(* IEC 61131-3 sources: generating_plc_code_with_llms/Code#1/Bard/third run, 21 files *)

(* ---- 14.st ---- *)
// 9.13s
// 2
FUNCTION FC1001(current_value: REAL, switching_value: REAL, hysteresis_percent: REAL): BOOL;
VAR
  previous_value: REAL;
  hysteresis_value: REAL;
  output_state: BOOL;

BEGIN

  // Initialize variables on first call
  IF NOT FC1001_initialized THEN
    previous_value := current_value;
    FC1001_initialized := TRUE;
  END_IF;

  // Calculate hysteresis value
  hysteresis_value := switching_value * hysteresis_percent / 100.0;

  // Determine output state based on current value and hysteresis
  IF current_value > switching_value + hysteresis_value THEN
    output_state := TRUE;
  ELSIF current_value < switching_value - hysteresis_value THEN
    output_state := FALSE;
  ELSE
    output_state := previous_value; // Maintain previous state to prevent fluttering
  END_IF;

  // Update previous value for next call
  previous_value := current_value;

  FC1001 := output_state;
END_FUNCTION

(* ---- 15.st ---- *)
// 12.79s
// 2
FUNCTION FC1002(E_A: BOOL, ultrasonic_presence: BOOL, P_HU: BOOL, P_AL: BOOL, P1: BOOL):
VAR
  monitoring_active: BOOL;
  presence_detected: BOOL;
  presence_timer: TIME;

BEGIN

  // Determine monitoring activation based on switch E_A
  monitoring_active := E_A;

  // Update presence_detected based on ultrasonic_presence and monitoring_active
  IF monitoring_active THEN
    IF ultrasonic_presence THEN
      presence_detected := TRUE;
    ELSIF NOT presence_detected THEN
      TOF(IN := TRUE, PT := #3000ms, Q := presence_timer);
    ELSE
      IF presence_timer.ET THEN
        presence_detected := FALSE;
      END_IF;
    END_IF;
  ELSE
    presence_detected := FALSE;
  END_IF;

  // Set output signals based on presence_detected and monitoring_active
  P_HU := monitoring_active AND presence_detected;
  P_AL := monitoring_active AND presence_detected AND presence_timer.ET;
  P1 := monitoring_active;

  FC1002 := (monitoring_active, presence_detected);
END_FUNCTION

(* ---- 18.st ---- *)
// 6.4s
// 2
FUNCTION FC1003(IN: REAL; IN_MIN: REAL; IN_MAX: REAL; OUT_MIN: REAL; OUT_MAX: REAL): REAL;

VAR
  range_factor: REAL;
  scaled_value: REAL;

BEGIN

  // Calculate range factor
  range_factor := (OUT_MAX - OUT_MIN) / (IN_MAX - IN_MIN);

  // Scale input value
  scaled_value := IN - IN_MIN;

  // Convert scaled value to output range
  FC1003 := scaled_value * range_factor + OUT_MIN;

  RETURN FC1003;
END_FUNCTION

(* ---- 19.st ---- *)
// 8.77s
// 2
FUNCTION_BLOCK FB1005

VAR
  START: BOOL;
  THICKNESS: BYTE;
  V_MAX: REAL;
  V_MIN: REAL;
  D_MAX: BYTE;
  D_MIN: BYTE;

  M_MAX: REAL;
  M_MIN: REAL;
  reject: BOOL;

BEGIN

  // Initialize variables
  M_MAX := 0.0;
  M_MIN := 0.0;
  reject := FALSE;

  // Read start signal
  START := SensorS1;

  // Read thickness
  THICKNESS := MD_1;

  // Check for new measurement
  IF START AND NOT reject THEN
    // Reset reject flag and minimum and maximum thickness values
    reject := FALSE;
    M_MAX := 0.0;
    M_MIN := 0.0;

    // Calculate thickness from laser measurements
    M_MAX := laser_measurement1 - laser_measurement2;

    // Check if thickness is outside tolerance
    IF M_MAX > V_MAX OR M_MAX < V_MIN THEN
      reject := TRUE;
      P1 := TRUE;
    END_IF;

    // Update minimum thickness value
    IF M_MIN = 0.0 OR M_MIN > M_MAX THEN
      M_MIN := M_MAX;
    END_IF;
  END_IF;

  // Write maximum thickness value to output
  D_MAX := INT(M_MAX);

  // Write minimum thickness value to output
  D_MIN := INT(M_MIN);

END_FUNCTION_BLOCK

(* ---- 21.st ---- *)
// 13.61s
// 2
FUNCTION_BLOCK BURNER

VAR
IN: BOOL;             // Start signal
OVER_TEMP: BOOL;      // Boiler thermostat protection
OIL_TEMP: BOOL;       // Oil temperature signal
STAGE2: BOOL;        // Second stage activation
RST: BOOL;            // Reset signal
STATUS: INT;       // Status output (110-Standby, 111-Startup, 112-Stage 1, 113-Stage 2)
ERROR: INT;         // Error output (0-No error, 1-Oil warming timeout, 2-Flame during pre-heat, ...)

internal_state: INT; // Internal state machine variable
timer_preheat: TIME;  // Timer for pre-heating
timer_prevent: TIME;  // Timer for pre-ventilation
timer_safety: TIME;   // Timer for flame safety
timer_post_ignit: TIME; // Timer for post-ignition delay
timer_stage2: TIME;   // Timer for stage 2 delay
timer_lockout: TIME;  // Timer for lockout

BEGIN

// Initialize variables
internal_state := 110; // Standby
timer_preheat := 0s;
timer_prevent := 0s;
timer_safety := 0s;
timer_post_ignit := 0s;
timer_stage2 := 0s;
timer_lockout := 0s;
STATUS := 110;
ERROR := 0;

// Main loop
WHILE TRUE DO

// Check for reset
IF RST THEN
  IF timer_lockout.ET THEN
    internal_state := 110;
    STATUS := 110;
    ERROR := 0;
  END_IF;
ELSE

  // Check overall conditions
  IF OVER_TEMP THEN
    internal_state := 110;
    STATUS := 110;
    ERROR := 9;
  ELSIF internal_state = 110 AND IN THEN
    internal_state := 111;
    STATUS := 111;
  END_IF;

  // State machine
  CASE internal_state OF
    111: // Startup sequence
      TOF(IN := TRUE, PT := #PRE_HEAT_TIME, Q := timer_preheat);
      IF OIL_TEMP AND timer_preheat.ET THEN
        internal_state := 112;
        STATUS := 112;
        timer_prevent := 0s;
      ELSIF timer_preheat.ET THEN
        internal_state := 110;
        STATUS := 110;
        ERROR := 1;
      END_IF;
    112: // Stage 1 operation
      TOF(IN := TRUE, PT := #PRE_VENTILATION_TIME, Q := timer_prevent);
      IF timer_prevent.ET THEN
        TOF(IN := TRUE, PT := #PRE_IGNITE_TIME, Q := timer_post_ignit);
        TOF(IN := TRUE, PT := #SAFETY_TIME, Q := timer_safety);
        IF (TIMER_IGNITION_ACTIVE) THEN
          ERROR := 2;
        ELSIF NOT TIMER_FLAME_DETECTED THEN
          ERROR := 4;
        ELSIF timer_safety.ET THEN
          internal_state := 112; // Restart ignition
          timer_post_ignit := 0s;
        ELSE
          TOF(IN := TRUE, PT := #POST_IGNITE_TIME, Q := timer_post_ignit);
          IF timer_post_ignit.ET AND NOT TIMER_FLAME_DETECTED THEN
            ERROR := 5;
          ELSE
            timer_stage2 := #STAGE2_DELAY;
          END_IF;
        END_IF;
      END_IF;
    113: // Stage 2 operation
      TOF(IN := TRUE, PT := timer_stage2, Q := timer_stage2);
      IF STAGE2 AND timer_stage2.ET THEN
        internal_state := 113; // Continue in stage 2
        timer_stage2 := 0s;
      ELSEIF NOT TIMER_FLAME_DETECTED OR MULTIPLE_IGNITION THEN
        internal_state := 112; // Restart ignition
// 23.8s
      ELSEIF NOT TIMER_FLAME_DETECTED OR MULTIPLE_IGNITION THEN
        internal_state := 112; // Restart ignition
        timer_post_ignit := 0s;
      END_IF;
    END_CASE;

    // Lockout timer
  TOF(IN := TRUE, PT := #LOCKOUT_TIME, Q := timer_lockout);

END_IF;

END_WHILE;

END_FUNCTION_BLOCK

(* ---- 1.st ---- *)
//5.95s
//3
PROGRAM MyProgram

VAR
  xAlarm1: BOOL;
  xAlarm2: BOOL;
  xAllOn: BOOL;
  xAllOff: BOOL;

BEGIN

  IF xAllOn THEN
    xAlarm1 := TRUE;
    xAlarm2 := TRUE;
  ELSIF xAllOff THEN
    xAlarm1 := FALSE;
    xAlarm2 := FALSE;
  ELSE
    // Process alarm conditions
  END_IF;

END_PROGRAM

(* ---- 10.st ---- *)
//7.98s
// 2
PROGRAM SigmoidFunction

VAR
  x: REAL;
  y: REAL;

FUNCTION Sigmoid(x: REAL): REAL;
  BEGIN
    y := 1.0 / (1.0 + Exp(-x));
    Sigmoid := y;
  END_FUNCTION;

BEGIN
  x := 1.0;
  y := Sigmoid(x);
END_PROGRAM

(* ---- 11.st ---- *)
//6.85s
// 2
PROGRAM SignFunction

VAR
  x: REAL;
  y: REAL;

FUNCTION Sign(x: REAL): REAL;
  BEGIN
    IF x > 0 THEN
      y := 1.0;
    ELSIF x < 0 THEN
      y := -1.0;
    ELSE
      y := 0.0;
    END_IF;
    Sign := y;
  END_FUNCTION;

BEGIN
  x := 1.0;
  y := Sign(x);
END_PROGRAM

(* ---- 12.st ---- *)
//8.86s
// 2
PROGRAM HyperbolicSine

VAR
x: REAL;
y: REAL;

FUNCTION Sinh(x: REAL): REAL;
BEGIN
y := (Exp(x) - Exp(-x)) / 2.0;
Sinh := y;
END_FUNCTION;

BEGIN
x := 1.0;
y := Sinh(x);
END_PROGRAM;

(* ---- 13.st ---- *)
//12.15s
// 2
PROGRAM NumberSearch

VAR
  numbers: ARRAY[0..99] OF INT;
  targetNumber: INT := 10;
  found: BOOL := FALSE;
  index: INT;

BEGIN

  // Initialize the list with random numbers
  FOR index := 0 TO 99 DO
    numbers[index] := RANDOM(1, 100);
  END_FOR;

  index := 0;

  REPEAT
    IF numbers[index] = targetNumber THEN
      found := TRUE;
      EXIT;
    END_IF;

    index := index + 1;
  UNTIL index = 100;

  // Handle the result
  IF found THEN
    WRITE_STRING('The number ' + STRING(targetNumber) + ' was found at index ' + STRING(index));
  ELSE
    WRITE_STRING('The number ' + STRING(targetNumber) + ' was not found in the list');
  END_IF;

END_PROGRAM

(* ---- 16.st ---- *)
//13.09s
// 2
PROGRAM TrafficLight

VAR
  North_green: BOOL;
  North_yellow: BOOL;
  North_red: BOOL;
  East_green: BOOL;
  East_yellow: BOOL;
  East_red: BOOL;
  timer: TIME;

BEGIN

  // Initialize all lights to red
  North_green := FALSE;
  North_yellow := FALSE;
  North_red := TRUE;
  East_green := FALSE;
  East_yellow := FALSE;
  East_red := TRUE;

  // Start the timer
  TON(IN := TRUE, PT := #10000ms, Q := timer);

  WHILE TRUE DO
    // Check the timer value and set the light signals accordingly
    IF timer.ET THEN
      // North light green
      North_green := TRUE;
      North_yellow := FALSE;
      North_red := FALSE;
      East_green := FALSE;
      East_yellow := FALSE;
      East_red := TRUE;

      // Wait for 5000ms
      DELAY(5000);

      // North light yellow
      North_green := FALSE;
      North_yellow := TRUE;
      North_red := FALSE;
      East_green := FALSE;
      East_yellow := FALSE;
      East_red := TRUE;

      // Wait for 500ms
      DELAY(500);

      // North light red, East light green
      North_green := FALSE;
      North_yellow := FALSE;
      North_red := TRUE;
      East_green := TRUE;
      East_yellow := FALSE;
      East_red := FALSE;

      // Wait for 4000ms
      DELAY(4000);

      // East light yellow
      North_green := FALSE;
      North_yellow := FALSE;
      North_red := TRUE;
      East_green := FALSE;
      East_yellow := TRUE;
      East_red := FALSE;

      // Wait for 500ms
      DELAY(500);

      // Reset the timer
      TOF(IN := timer.Q, PT := #10000ms, Q := timer);
    END_IF;
  END_WHILE;

END_PROGRAM

(* ---- 17.st ---- *)
//11.4s
// 2
PROGRAM WeatherStation

VAR
  temperatureAnalogValue: INT; // Temperature analog input value
  temperaturePercent: REAL; // Temperature converted to percent
  humidity: INT; // Humidity analog input value
  humidityPercent: REAL; // Humidity converted to percent
  temperatureText: STRING(10); // Text representation of temperature
  overallText: STRING(10); // Overall assessment of temperature and humidity

BEGIN

  // Read temperature analog value
  temperatureAnalogValue := ReadAnalogInput(TemperatureAnalogInputChannel);

  // Convert temperature analog value to percent
  temperaturePercent := REAL(temperatureAnalogValue) / 32767.0 * 100.0;

  // Evaluate temperature and set temperature text
  IF temperaturePercent < 18.0 THEN
    temperatureText := 'Cold';
  ELSIF temperaturePercent <= 25.0 THEN
    temperatureText := 'Opt';
  ELSE
    temperatureText := 'Hot';
  END_IF;

  // Read humidity analog value
  humidity := ReadAnalogInput(HumidityAnalogInputChannel);

  // Convert humidity analog value to percent
  humidityPercent := REAL(humidity) / 32767.0 * 100.0;

  // Evaluate humidity and temperature
  IF 40.0 <= humidityPercent <= 75.0 AND 18.0 <= temperaturePercent <= 25.0 THEN
    overallText := 'Opt';
  ELSE
    overallText := 'Temp. OK';
  END_IF;

  // Display temperature and humidity
  WRITE_STRING('Temperature: ' + STRING(temperaturePercent) + '% - ' + temperatureText);
  WRITE_STRING('Humidity: ' + STRING(humidityPercent) + '% - ' + overallText);

END_PROGRAM

(* ---- 2.st ---- *)
//4.63s
//2
PROGRAM BinomialCoefficient

VAR
  n: INT;
  k: INT;
  result: INT;

BEGIN

  IF k > n OR k < 0 THEN
    result := 0;
  ELSIF k = 0 OR k = n THEN
    result := 1;
  ELSE
    result := BinomialCoefficient(n - 1, k - 1) + BinomialCoefficient(n - 1, k);
  END_IF;
END_PROGRAM

(* ---- 20.st ---- *)
// 8.08s
// 2
PROGRAM Interlock

VAR
  I1: BOOL;
  I2: BOOL;
  Q1: BOOL;
  Q2: BOOL;
  Q1Timer: TIME;
  Q2Timer: TIME;

BEGIN

  // Initialize timers
  Q1Timer := 0.0s;
  Q2Timer := 0.0s;

  WHILE TRUE DO
    // Check input I1
    IF I1 THEN
      // Enable timer for Q1
      TOF(IN := TRUE, PT := #TL, Q := Q1Timer);

      // Set output Q1
      Q1 := TRUE;

      // Reset output Q2
      Q2 := FALSE;

      // Clear Q2 timer
      Q2Timer := 0.0s;
    END_IF;

    // Check input I2
    IF I2 THEN
      // Enable timer for Q2
      TOF(IN := TRUE, PT := #TL, Q := Q2Timer);

      // Set output Q2
      Q2 := TRUE;

      // Reset output Q1
      Q1 := FALSE;

      // Clear Q1 timer
      Q1Timer := 0.0s;
    END_IF;

    // Check if Q2 can be enabled
    IF Q2Timer > TL AND NOT Q2 THEN
      // Enable Q2
      Q2Timer := 0.0s;

      Q2 := TRUE;
    END_IF;

    // Check if Q1 can be enabled
    IF Q1Timer > TL AND NOT Q1 THEN
      // Enable Q1
      Q1Timer := 0.0s;

      Q1 := TRUE;
    END_IF;
  END_WHILE;

END_PROGRAM

(* ---- 3.st ---- *)
//10.15s
// 2
PROGRAM Fibonacci

VAR
  n: INT;
  result: INT;

FUNCTION Fibonacci(n: INT): INT;
VAR
  a: INT;
  b: INT;
  i: INT;

BEGIN
  a := 0;
  b := 1;

  FOR i := 1 TO n DO
    result := a + b;
    a := b;
    b := result;
  END_FOR;

  Fibonacci := result;
END_FUNCTION;

BEGIN
  n := 10;
  result := Fibonacci(n);
END_PROGRAM

(* ---- 4.st ---- *)
//7.39s
// 2
PROGRAM FillLevelCheck

VAR
  fillLevelAnalogValue: INT;
  fillLevelPercent: REAL;
  lowLevelOutput: BOOL;
  okLevelOutput: BOOL;
  highLevelOutput: BOOL;
  warningHornOutput: BOOL;

BEGIN

  // Read the fill level analog value
  fillLevelAnalogValue := ReadAnalogInput(AnalogInputChannel);

  // Convert the analog value to a percentage
  fillLevelPercent := REAL(fillLevelAnalogValue) / 32767.0 * 100.0;

  // Check the fill level and set the output variables accordingly
  CASE fillLevelPercent OF
    0.0 TO 1.0:
      lowLevelOutput := TRUE;
      okLevelOutput := FALSE;
      highLevelOutput := FALSE;
      warningHornOutput := TRUE;
    1.0 TO 90.0:
      lowLevelOutput := FALSE;
      okLevelOutput := TRUE;
      highLevelOutput := FALSE;
      warningHornOutput := FALSE;
    90.0 TO 100.0:
      lowLevelOutput := FALSE;
      okLevelOutput := FALSE;
      highLevelOutput := TRUE;
      warningHornOutput := FALSE;
    ELSE:
      // Invalid fill level
  END_CASE;

  // Write the output variables to the outputs
  WriteDigitalOutput(LowLevelOutputChannel, lowLevelOutput);
  WriteDigitalOutput(OkLevelOutputChannel, okLevelOutput);
  WriteDigitalOutput(HighLevelOutputChannel, highLevelOutput);
  WriteDigitalOutput(WarningHornOutputChannel, warningHornOutput);

END_PROGRAM

(* ---- 5.st ---- *)
//10.45s
// 2
PROGRAM GateController

VAR
  Start_Loop: BOOL;
  Gate_Open: BOOL;
  App_Or_Car_Sensed: BOOL;
  Auth_String: STRING(10);
  One_Hour_Timer: TIME;

BEGIN

  // Check if the start loop signal is active
  IF Start_Loop THEN
    // Start the one-hour timer
    TON(IN := TRUE, PT := #1H, Q := One_Hour_Timer);

    // Check if the gate is open and the timer has timed out
    IF Gate_Open AND One_Hour_Timer.ET THEN
      // Close the gate
      Gate_Open := FALSE;
    END_IF;

    // Check if the app or car is sensed and the authentication string matches
    IF App_Or_Car_Sensed AND Auth_String = 'my_defined_str' THEN
      // Open the gate
      Gate_Open := TRUE;
    END_IF;
  ELSE
    // Stop the one-hour timer
    TOF(IN := One_Hour_Timer.Q, PT := #1H, Q := One_Hour_Timer);
  END_IF;

END_PROGRAM

(* ---- 6.st ---- *)
//12.33s
// 2 nicht alle Variablen deklariert
PROGRAM CraneLift

VAR
  diConvTop: BOOL; // Light barrier for top conveyor belt
  diConvBottom: BOOL; // Light barrier for bottom conveyor belt
  doConvTop: BOOL; // Control signal for top conveyor belt
  doConvBottom: BOOL; // Control signal for bottom conveyor belt
  doLiftTop: BOOL; // Control signal for lift to top position
  doLiftBottom: BOOL; // Control signal for lift to bottom position
  doLiftUnload: BOOL; // Control signal for lift to unload position
  diLiftTop: BOOL; // Sensor indicating lift is in top position
  diLiftBottom: BOOL; // Sensor indicating lift is in bottom position
  diLiftUnload: BOOL; // Sensor indicating lift is in unload position
  doConvLift: BOOL; // Control signal for lift conveyor belt
  diBoxLift: BOOL; // Sensor indicating box is on lift

BEGIN

  // Handle top conveyor belt
  IF diConvTop THEN
    doConvTop := FALSE; // Stop top conveyor belt
    RequestLift('top'); // Request lift to top position
  ELSE
    doConvTop := TRUE; // Start top conveyor belt
  END_IF;

  // Handle bottom conveyor belt
  IF diConvBottom THEN
    doConvBottom := FALSE; // Stop bottom conveyor belt
    RequestLift('bottom'); // Request lift to bottom position
  ELSE
    doConvBottom := TRUE; // Start bottom conveyor belt
  END_IF;

  // Move lift to requested position
  IF liftRequested AND NOT liftAtPosition THEN
    IF requestedPosition = 'top' THEN
      doLiftTop := TRUE;
      doLiftBottom := FALSE;
    ELSIF requestedPosition = 'bottom' THEN
      doLiftTop := FALSE;
      doLiftBottom := TRUE;
    END_IF;
  ELSE
    doLiftTop := FALSE;
    doLiftBottom := FALSE;
  END_IF;

  // Handle lift conveyor belt
  IF liftAtPosition AND diBoxLift THEN
    doConvLift := TRUE; // Start lift conveyor belt
  ELSE
    doConvLift := FALSE; // Stop lift conveyor belt
  END_IF;

  // Move lift to unload position
  IF liftAtPosition AND diBoxLift THEN
    doLiftUnload := TRUE;
  ELSE
    doLiftUnload := FALSE;
  END_IF;

  // Unload box
  IF liftAtPosition AND diBoxLift AND diLiftUnload THEN
    UnloadBox();
    liftRequested := FALSE;
  END_IF;

END_PROGRAM

(* ---- 7.st ---- *)
//6.78s
// 2
PROGRAM Crane

(* Define constants *)
CONST
  NUM_LOAD_RECEPTORS: INT := 5;
  MAX_LOAD_VALUE: INT := 32767;

(* Define variables *)
VAR
  loadValues: ARRAY[0..NUM_LOAD_RECEPTORS-1] OF INT;
  totalLoad: INT;
  averageLoad: REAL;

BEGIN

(* Read load values from analog inputs *)
FOR i := 0 TO NUM_LOAD_RECEPTORS-1 DO
  loadValues[i] := ReadAnalogInput(AnalogInputChannel + i);
END_FOR;

(* Calculate total load *)
totalLoad := 0;
FOR i := 0 TO NUM_LOAD_RECEPTORS-1 DO
  totalLoad := totalLoad + loadValues[i];
END_FOR;

(* Calculate average load *)
averageLoad := REAL(totalLoad) / NUM_LOAD_RECEPTORS;

(* Process average load *)
IF averageLoad > MAX_LOAD_VALUE / 2 THEN
  // Overloaded condition
ELSIF averageLoad < MAX_LOAD_VALUE / 4 THEN
  // Underloaded condition
ELSE
  // Normal load condition
END_IF;

END_PROGRAM

(* ---- 8.st ---- *)
//9.09s
// 2
PROGRAM LambertW

VAR
  x: REAL;
  w: REAL;

FUNCTION LambertW(x: REAL): REAL;
  VAR
    epsilon: REAL;
    y: REAL;
    oldY: REAL;
    i: INT;

  BEGIN
    epsilon := 0.0001;
    y := x;
    oldY := 0.0;
    i := 0;

    WHILE ABS(y - oldY) > epsilon DO
      i := i + 1;
      oldY := y;
      y := Exp(y) * (1.0 + y);
    END_WHILE;

    LambertW := y;
  END_FUNCTION;

BEGIN
  x := 0.5;
  w := LambertW(x);
END_PROGRAM

(* ---- 9.st ---- *)
//7.66s
// 2
PROGRAM LeapYearChecker

VAR
  YEAR: INT;
  isLeapYear: BOOL;

BEGIN

  // Check if the year is divisible by 4
  IF YEAR MOD 4 = 0 THEN
    // Check if the year is also divisible by 100
    IF YEAR MOD 100 = 0 THEN
      // Check if the year is also divisible by 400
      IF YEAR MOD 400 = 0 THEN
        isLeapYear := TRUE;
      ELSE
        isLeapYear := FALSE;
      END_IF;
    ELSE
      isLeapYear := TRUE;
    END_IF;
  ELSE
    isLeapYear := FALSE;
  END_IF;

  // Output the result
  IF isLeapYear THEN
    WRITE_STRING('The year ' + STRING(YEAR) + ' is a leap year.');
  ELSE
    WRITE_STRING('The year ' + STRING(YEAR) + ' is not a leap year.');
  END_IF;

END_PROGRAM
